FUNCTION_BLOCK FB_TEST_CheckPartGood EXTENDS FB_Test
VAR
END_VAR

METHOD Execute : ST_TestResults
VAR
	MockStatus		: ST_PartStatus;
	fbCell			: FB_Cell;
	testExpected	: BOOL;
	testResult		: BOOL;
END_VAR
MockStatus.bBarcodeStatus := TRUE;
MockStatus.bCapperStatus := TRUE;
MockStatus.bFillerStatus := TRUE;
MockStatus.bWeightStatus := TRUE;

testExpected := TRUE;
testResult := fbCell.CheckPart(MockStatus);

Execute := AssertEquals(
	testExpected, 
	testResult, 
	'CheckPart Part status mismatch.'
);
END_METHOD

END_FUNCTION_BLOCK

(* stored: Version 1.1.0.1, ProductVersion 3.1.4026.7
   POU FB_TEST_CheckPartGood: Id {5db17b90-6099-47d9-989c-c5b0fd1881b9}, SpecialFunc None
   Method Execute: Id {3f0f40f1-6564-4c24-b10b-2596e7cc6c4e} *)
